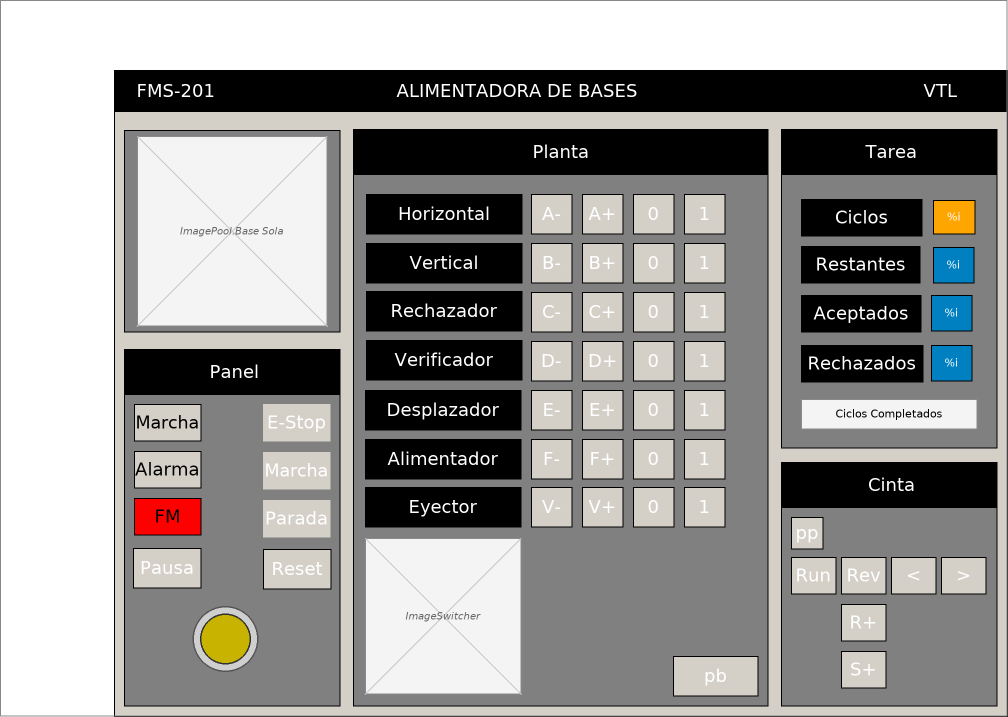
VISUALIZATION Visualization  // 1008x717
    Rectangle (114,111 894x606)
    Rectangle (781,174 216x274)
    Rectangle (353,174 415x532)
    Rectangle (353,129 415x45)
    Label (353,131 416x42), "Planta"
    Rectangle (781,129 216x45)
    Label (831,134 121x36), "Tarea"
    Progressbar (801,399 176x30), "Ciclos Completados", variable: MAIN.test_pieza.Aceptados
    RoundedRectangle (366,194 156x40), "Horizontal"
    Textfield (933,200 42x34), "%i", text variable: MAIN.Estacion.CiclosSolicitados
        OnMouseDown: write MAIN.Estacion.CiclosSolicitados via VisuDialogs.Numpad, min 1, max 10
    RoundedRectangle (801,199 121x37), "Ciclos"
    RoundedRectangle (801,246 119x37), "Restantes"
    RoundedRectangle (801,295 120x37), "Aceptados"
    RoundedRectangle (801,345 122x37), "Rechazados"
    Textfield (933,247 41x36), "%i", text variable: MAIN.Estacion.CiclosPendientes
    Textfield (931,295 41x36), "%i", text variable: MAIN.Estacion.CiclosAceptados
    Textfield (931,345 41x36), "%i", text variable: MAIN.Estacion.CiclosRechazados
    RoundedRectangle (582,243 41x40), "B+", colour toggle: MAIN.Estacion.Descargador_baja
        toggle MAIN.Estacion.Descargador_baja
    Rectangle (781,507 216x199)
    Rectangle (781,462 216x45)
    Label (831,467 121x36), "Cinta"
    Rectangle (124,130 216x202)
    Rectangle (124,394 216x312)
    Rectangle (124,349 216x45)
    Label (174,354 121x36), "Panel"
    Rectangle (114,70 894x41)
    Label (114,71 893x40), "FMS-201 ALIMENTADORA DE BASES VTL"
    RoundedRectangle (366,243 156x40), "Vertical"
    RoundedRectangle (582,194 41x40), "A+", colour toggle: MAIN.Estacion.Descargador_adelante
        tap MAIN.Estacion.Descargador_adelante
    RoundedRectangle (582,292 41x40), "C+", colour toggle: MAIN.Estacion.Rechazador_adelante
        tap MAIN.Estacion.Rechazador_adelante
    RoundedRectangle (582,341 41x40), "D+", colour toggle: MAIN.Estacion.Verificador_baja
        tap MAIN.Estacion.Verificador_baja
    RoundedRectangle (582,390 41x40), "E+", colour toggle: MAIN.Estacion.Desplazador_adelante
        tap MAIN.Estacion.Desplazador_adelante
    RoundedRectangle (582,439 41x40), "F+", colour toggle: MAIN.Estacion.Alimentador_adelante
        tap MAIN.Estacion.Alimentador_adelante
    RoundedRectangle (582,487 41x40), "V+", colour toggle: MAIN.Estacion.Eyector_succiona
        toggle MAIN.Estacion.Eyector_succiona
    RoundedRectangle (366,291 156x40), "Rechazador"
    RoundedRectangle (366,340 156x40), "Verificador"
    RoundedRectangle (365,390 156x40), "Desplazador"
    RoundedRectangle (365,439 156x40), "Alimentador"
    RoundedRectangle (365,487 156x40), "Eyector"
    RoundedRectangle (531,194 41x40), "A-", colour toggle: MAIN.Estacion.Descargador_atras
        tap MAIN.Estacion.Descargador_atras
    RoundedRectangle (633,194 41x40), "0", colour toggle: MAIN.Estacion.Horizontal_descargador_detras
    RoundedRectangle (684,194 41x40), "1", colour toggle: MAIN.Estacion.Horizontal_descargador_delante
    RoundedRectangle (633,243 41x40), "0", colour toggle: MAIN.Estacion.Vertical_descargador_arriba
        tap MAIN.Estacion.Vertical_descargador_arriba
    RoundedRectangle (684,243 41x40), "1", colour toggle: MAIN.Estacion.Vertical_descargador_abajo
        tap MAIN.Estacion.Vertical_descargador_abajo
    RoundedRectangle (633,292 41x40), "0"
    RoundedRectangle (633,341 41x40), "0", colour toggle: MAIN.Estacion.Verificador_arriba
        tap MAIN.Estacion.Verificador_arriba
    RoundedRectangle (633,390 41x40), "0", colour toggle: MAIN.Estacion.Desplazador_detras
        tap MAIN.Estacion.Desplazador_detras
    RoundedRectangle (633,439 41x40), "0", colour toggle: MAIN.Estacion.Alimentador_detras
        tap MAIN.Estacion.Alimentador_detras
    RoundedRectangle (633,487 41x40), "0"
    RoundedRectangle (684,292 41x40), "1"
    RoundedRectangle (684,341 41x40), "1", colour toggle: MAIN.Estacion.Verificador_abajo
        tap MAIN.Estacion.Verificador_abajo
    RoundedRectangle (684,390 41x40), "1"
    RoundedRectangle (684,439 41x40), "1", colour toggle: MAIN.Estacion.Alimentador_delante
        tap MAIN.Estacion.Alimentador_delante
    RoundedRectangle (684,487 41x40), "1", colour toggle: MAIN.Estacion.Vacio_obtenido_vacuostato_descargador
        tap MAIN.Estacion.Vacio_obtenido_vacuostato_descargador
    RoundedRectangle (531,243 41x40), "B-"
    RoundedRectangle (531,292 41x40), "C-"
    RoundedRectangle (531,341 41x40), "D-"
    RoundedRectangle (531,390 41x40), "E-"
    RoundedRectangle (531,439 41x40), "F-"
    RoundedRectangle (531,487 41x40), "V-"
    RoundedRectangle (673,656 85x40), "pb", colour toggle: MAIN.Estacion.Base_en_Alimentador
        tap MAIN.Estacion.Base_en_Alimentador
    RoundedRectangle (134,498 67x37), "FM", colour toggle: MAIN.Estacion.Lampara_falta_material
        tap MAIN.Estacion.Lampara_falta_material
    RoundedRectangle (791,517 32x32), "pp", colour toggle: MAIN.Estacion.Presencia_pale
        tap MAIN.Estacion.Presencia_pale
    RoundedRectangle (941,557 45x37), ">", colour toggle: MAIN.Estacion.Activa_marcha_motor_cinta
        tap MAIN.Estacion.Activa_marcha_motor_cinta
    RoundedRectangle (891,557 45x37), "<", colour toggle: MAIN.Estacion.Invierte_marcha_motor_cinta
        toggle MAIN.Estacion.Invierte_marcha_motor_cinta
    RoundedRectangle (791,557 45x37), "Run", colour toggle: MAIN.Estacion.Activa_marcha_motor_cinta
    RoundedRectangle (841,557 45x37), "Rev", colour toggle: MAIN.Estacion.Invierte_marcha_motor_cinta
    RoundedRectangle (841,604 45x37), "R+", colour toggle: MAIN.Estacion.Retenedor_pale_baja
        toggle MAIN.Estacion.Retenedor_pale_baja
    RoundedRectangle (841,651 45x37), "S+", colour toggle: MAIN.Estacion.Separador_pale_sube
        toggle MAIN.Estacion.Separador_pale_sube
    RoundedRectangle (263,404 67x37), "E-Stop", colour toggle: MAIN.Estacion.Pulsador_parada_emergencia
        tap MAIN.Estacion.Pulsador_parada_emergencia
    RoundedRectangle (263,452 67x37), "Marcha", colour toggle: MAIN.Estacion.Pulsador_marcha
        tap MAIN.Estacion.Pulsador_marcha
    RoundedRectangle (263,500 67x37), "Parada", colour toggle: MAIN.Estacion.Pulsador_parada_NC
        tap MAIN.Estacion.Pulsador_parada_NC
    RoundedRectangle (134,451 67x37), "Alarma", colour toggle: MAIN.Estacion.Lampara_alarma
        tap MAIN.Estacion.Lampara_alarma
    RoundedRectangle (134,404 67x37), "Marcha", colour toggle: MAIN.Estacion.Lampara_marcha
        tap MAIN.Estacion.Lampara_marcha
    Image (137,136 190x190), image: ImagePool.Base Sola
    Lamp1 (187,601 77x76), variable: MAIN.test_pieza.Lampara_falta_material, style: Lamp-Lamp1-Yellow
    ImageSwitcher (365,538 156x156), variable: MAIN.Estacion.pieza_ok, background image: ImagePool.Base OK, image: ImagePool.Base No OK, behaviour: TOGGLE
    RoundedRectangle (133,548 68x40), "Pausa", text variable: MAIN.Estacion.EstadoPausa, colour toggle: MAIN.Estacion.EstadoPausaMAIN.Estacion.EstadoPausa
        tap MAIN.Estacion.EstadoPausa
    RoundedRectangle (263,549 68x40), "Reset", text variable: MAIN.Estacion.EstadoReinicia, colour toggle: MAIN.Estacion.EstadoReinicia
        tap MAIN.Estacion.EstadoReinicia
END_VISUALIZATION

(* stored: Version 1.1.0.1, ProductVersion 3.1.4024.12
   Visu Visualization: Id {bc3923f8-cf4b-42b1-a17b-2f6c76ade0ae} *)
